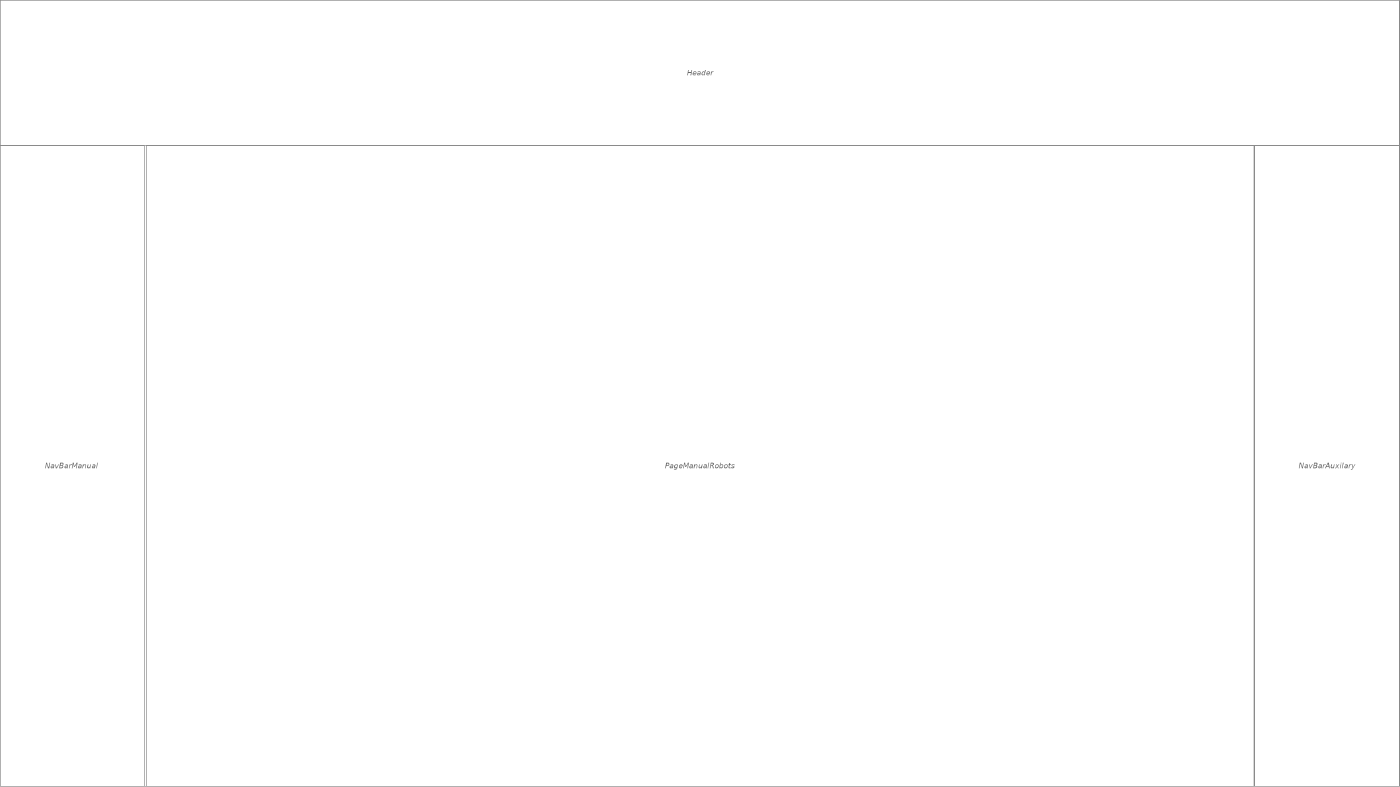
VISUALIZATION Main  // 1920x1080
    Frame (0,0 1920x200)
        shows Header(sMachineName := PRG_VisuControl.fbVisuControl.sMachineName, sSoftwareVersion := PRG_VisuControl.fbVisuControl.sSoftwareVersion, eMachineState := PRG_MachineControl.fbMachineControler.eMachineState, sCurrentRecipe := PRG_VisuControl.fbVisuControl.sCurrentRecipe, sCurrentUser := PRG_VisuControl.fbVisuControl.sCurrentUser, iActiveCriticals := PRG_VisuControl.fbVisuControl.iActiveCriticals, iActvieErrors := PRG_VisuControl.fbVisuControl.iActvieErrors, iActiveWarrnings := PRG_VisuControl.fbVisuControl.iActiveWarrnings, sCurrentDate := PRG_VisuControl.fbVisuControl.sCurrentDate, sCurrentTime := PRG_VisuControl.fbVisuControl.sCurrentTime)
    Frame (1720,199 200x880)
        shows NavBarAuxilary(btnAlarms := PRG_VisuControl.fbVisuControl.btnAlarms, btnRecipes := PRG_VisuControl.fbVisuControl.btnRecipes, btnDoorLock := PRG_VisuControl.fbVisuControl.btnLights, btnLogIn := PRG_VisuControl.fbVisuControl.btnLogIn, btnLogOut := PRG_VisuControl.fbVisuControl.btnLogOut, btnHmiClose := PRG_VisuControl.fbVisuControl.btnHmiClose, sCloseHMIFileName := PRG_VisuControl.fbVisuControl.sCloseHMIFileName, sCloseHMIParameters := PRG_VisuControl.fbVisuControl.sCloseHMIParameters, bVisNotInit := PRG_VisuControl.fbVisuControl.bVisNotInit, bVisHmiCLose := PRG_VisuControl.fbVisuControl.bVisHmiClose, bVisLogIn := PRG_VisuControl.fbVisuControl.bVisLogIn, bVisLogOut := PRG_VisuControl.fbVisuControl.bVisLogOut, bDoorLockDisabled := PRG_VisuControl.fbVisuControl.btnLights, bDoorLockInvisible := PRG_VisuControl.fbVisuControl.btnLights)
    Frame (200,199 1520x880)
        shows PageManualRobots(btnPrevious := PRG_VisuControl.fbVisuControl.btnPrevious, btnNext := PRG_VisuControl.fbVisuControl.btnNext, bPreviousInvisible := PRG_VisuControl.fbVisuControl.bPreviousInvisible, bNextInvisible := PRG_VisuControl.fbVisuControl.bNextInvisible, stRobotEmpty := PRG_VisuControl.fbVisuControl.arrRobotFrameEmpty[PRG_VisuControl.fbVisuControl.iSelectedRobotPageIndex], stRobot := PRG_VisuControl.fbVisuControl.arrRobotFrame[PRG_VisuControl.fbVisuControl.iSelectedRobotPageIndex], iRobotSelectedPageIndex := PRG_VisuControl.fbVisuControl.iSelectedRobotPageIndex, iRobotTotalPageIndex := PRG_VisuControl.fbVisuControl.iRobotPageIndex)
    Frame (-2,199 200x880)
        shows NavBarManual(btnAutoMode := PRG_VisuControl.fbVisuControl.btnAuto, btnCylinders := PRG_VisuControl.fbVisuControl.btnManualCylinder, btnMotors := PRG_VisuControl.fbVisuControl.btnManualAxis, btnSafety := PRG_VisuControl.fbVisuControl.btnManualSafety, btnInputs := PRG_VisuControl.fbVisuControl.btnManualInputs, btnOutputs := PRG_VisuControl.fbVisuControl.btnManualOutputs, btnOthers := PRG_VisuControl.fbVisuControl.btnManualOthers, btnAbort := PRG_VisuControl.fbVisuControl.btnAbort, btnRobots := PRG_VisuControl.fbVisuControl.btnManualRobots)
END_VISUALIZATION

(* stored: Version 1.1.0.1, ProductVersion 3.1.4024.9
   Visu Main: Id {4c31c11e-56ef-4c33-8502-9b678708e8e5} *)
